# EPICS substitutions: synApps_6_1/support/motor-R7-1/modules/motorMclennan/iocs/mclennanIOC/iocBoot/iocMclennan/PM304.substitutions
file "$(MOTOR)/db/motor.db"
{
pattern
{P,         N,     M,         DTYP,           C, S, DESC,          EGU,    DIR,	VELO, VBAS, ACCL, BDST, BVEL, BACC, MRES, PREC, DHLM, DLLM, INIT}
{mclennan:, 1, "m$(N)", "Mclennan PM304",     0, 0, "motor $(N)", degrees, Pos, 10,    0.,   1.,   0,    1,    .2,   1e-3, 3,    100,  -100, ""}
}
